KUKA KRL program: amm_warning.src

&ACCESS RV
&REL 4
&PARAM EDITMASK = *
&PARAM TEMPLATE = C:\KRC\Roboter\Template\vorgabe
DEF AMM_warning(FI_tReaction :IN)
DECL TYPMillReaction FI_tReaction
DECL INT FI_nNumber

; for example
  ;Stop Robot
    BRAKE
  ;Stop Process
    milling_abort()

  AMM_message(106,#DIALOG,gnMillMsgAnswer )
  IF (gnMillMsgAnswer == 1) THEN
     ; do nothing
  ENDIF
  ;Start Process
    UP_Start(FALSE)

;FOLD User Actions

;ENDFOLD

END
